FUNCTION_BLOCK Wp (* Composite Function Block Type *)
  (* Standard: 61499-2 *)
  (* Version 0.0, 7/15/2016, Andrei, nxtControl GmbH, template *)
  PACKAGE Main;
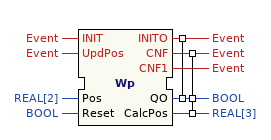
  EVENT_INPUT
    INIT; (* Initialization Request *)
    UpdPos; (* Normal Execution Request *)
  END_EVENT
  EVENT_OUTPUT
    INITO WITH QO; (* Initialization Confirm *)
    CNF WITH QO, CalcPos; (* Execution Confirmation *)
    CNF1; (* Execution Confirmation *)
  END_EVENT
  VAR_INPUT
    Pos : ARRAY [0..1] OF REAL; (* Input event qualifier *)
    Reset : BOOL;
  END_VAR
  VAR_OUTPUT
    QO : BOOL; (* Output event qualifier *)
    CalcPos : ARRAY [0..2] OF REAL; (* Output event qualifier *)
  END_VAR
  FBS
    FB1 : E_PERMIT;
    FB2 : ChangeDetect;
    FB3 : integEC(minValue := 0.0, maxValue := 10.0, pv1 := 20.0, cycleTime := 0.02, preTrip := 0.0, integType := 0, sp := 100.0, tBase1 := 1.0, tBase2 := 4.0, useLimits := TRUE, pv2 := 0.0, inv1 := FALSE, inv2 := FALSE);
    FB5 : NOT_42C76073DCEB1A7A; {SET_ATTRIBUTE(Configuration.GenericFBType.InterfaceParams, Runtime.Standard#CNT:=1;OUT${CNT$}:BOOL)}
    FB6 : ADD_1990CFD1468AAE4A6; {SET_ATTRIBUTE(Configuration.GenericFBType.InterfaceParams, Runtime.Standard#CNT:=2;IN${CNT$}:LREAL)}
    FB9 : ChangeDetect;
    FB7 : Demux;
    FB4 : E_PERMIT;
    FB8 : Muxer;
    FB10 : ADDER;
  END_FBS
  EVENT_CONNECTIONS
    FB1.EO TO FB3.C_CYCLE;
    UpdPos TO FB5.REQ;
    FB5.CNF TO FB1.EI;
    FB3.CNF TO FB10.REQ;
    FB7.CNF TO FB2.REQ;
    FB7.CNF TO FB9.REQ;
    UpdPos TO FB7.REQ;
    FB10.CNF TO FB8.REQ;
    FB8.CNF TO CNF1;
    FB4.EO TO FB3.RESET;
    FB5.CNF TO FB4.EI;
    INIT TO FB3.INIT;
  END_CONNECTIONS
  DATA_CONNECTIONS
    FB5.OUT1 TO FB1.PERMIT;
    FB3.out TO FB10.In2;
    Reset TO FB5.IN1;
    FB7.X TO FB2.INP;
    FB7.Y TO FB9.INP;
    Pos TO FB7.InData;
    FB7.Y TO FB10.In1;
    FB10.Out TO FB8.Y;
    FB7.X TO FB8.X;
    FB8.DataOut TO CalcPos;
    Reset TO FB4.PERMIT;
    FB3.out TO FB8.Ye;
  END_CONNECTIONS
END_FUNCTION_BLOCK
